{attribute 'pack_mode' := '1'}
    {attribute 'OPC.UA.DA' := '1'}
    {attribute 'OPC.UA.DA.StructuredType' := '1'}
    (*
    ST_RW_PlcDeviceStatus_HMI_IgnitionExp
    ==================================================
    Generated from Ignition UDT: RW_PLC_Device_Status
    Total tags: 3
    Generated on: 2025-09-15 12:47:18
    *)
    TYPE ST_RW_PlcDeviceStatus_HMI_IgnitionExp :
    STRUCT
        {attribute 'OPC.UA.DA' := '1'}
        {attribute 'OPC.UA.DA.Access' := '1'}
        Name : STRING := '';		// Read-only tag
        {attribute 'OPC.UA.DA' := '1'}
        {attribute 'OPC.UA.DA.Access' := '1'}
        IPAddress : STRING := '';		// Read-only tag
        {attribute 'OPC.UA.DA' := '1'}
        {attribute 'OPC.UA.DA.Access' := '1'}
        State : DINT := 0;		// Read-only tag
    END_STRUCT
    END_TYPE

(* stored: Version 1.1.0.1
   DUT ST_RW_PlcDeviceStatus_HMI_IgnitionExp: Id {3516e07d-4675-48a5-abbd-2eeebc1ff0f6} *)
